INTERFACE I_AveCorredora

METHOD Correr : BOOL
END_METHOD

END_INTERFACE

(* stored: Version 1.1.0.1, ProductVersion 3.1.4024.12
   Itf I_AveCorredora: Id {50283ac5-eda6-4d5d-b3cb-87fde271d92b}
   Method Correr: Id {7cc4fb4f-861b-42ff-bd9c-5aa1137519b6} *)
